// LS Electric XG5000 project: JG 비젼 프로그램
// PLC LSPLC
// module base 0 slot 0: 입출력 모듈:XBM-DN32H (DC 24V입력/TR 출력, 32점)

PROGRAM NewProgram (task: 스캔 프로그램)

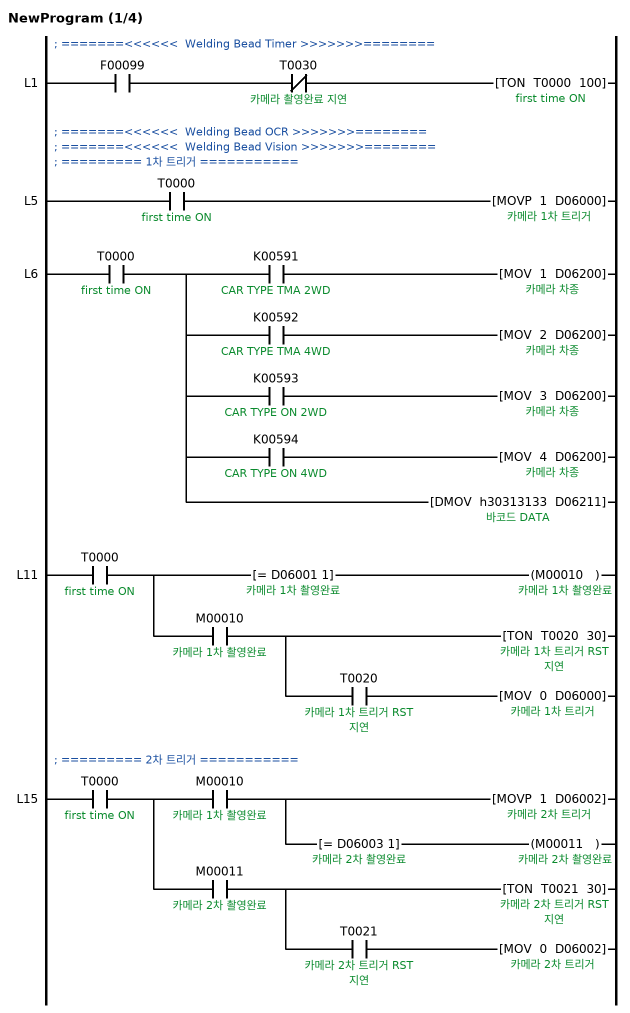
// =======<<<<<<  Welding Bead Timer >>>>>>>========
; L1
LOAD      F00099
AND NOT   T0030	// 카메라 촬영완료 지연
TON       T0000 100	// first time ON
// =======<<<<<<  Welding Bead OCR >>>>>>>========
// =======<<<<<<  Welding Bead Vision >>>>>>>========
// ========= 1차 트리거 ===========
; L5
LOAD      T0000	// first time ON
MOVP      1 D06000	// 카메라 1차 트리거
; L6
LOAD      T0000	// first time ON
MPUSH
AND       K00591	// CAR TYPE TMA 2WD
MOV       1 D06200	// 카메라 차종
MLOAD
AND       K00592	// CAR TYPE TMA 4WD
MOV       2 D06200	// 카메라 차종
MLOAD
AND       K00593	// CAR TYPE ON 2WD
MOV       3 D06200	// 카메라 차종
MLOAD
AND       K00594	// CAR TYPE ON 4WD
MOV       4 D06200	// 카메라 차종
MPOP
DMOV      h30313133 D06211	// 바코드 DATA
; L11
LOAD      T0000	// first time ON
MPUSH
AND=      D06001 1	// 카메라 1차 촬영완료
OUT       M00010	// 카메라 1차 촬영완료
MPOP
AND       M00010	// 카메라 1차 촬영완료
TON       T0020 30	// 카메라 1차 트리거 RST 지연
AND       T0020	// 카메라 1차 트리거 RST 지연
MOV       0 D06000	// 카메라 1차 트리거
// ========= 2차 트리거 ===========
; L15
LOAD      T0000	// first time ON
MPUSH
AND       M00010	// 카메라 1차 촬영완료
MOVP      1 D06002	// 카메라 2차 트리거
AND=      D06003 1	// 카메라 2차 촬영완료
OUT       M00011	// 카메라 2차 촬영완료
MPOP
AND       M00011	// 카메라 2차 촬영완료
TON       T0021 30	// 카메라 2차 트리거 RST 지연
AND       T0021	// 카메라 2차 트리거 RST 지연
MOV       0 D06002	// 카메라 2차 트리거

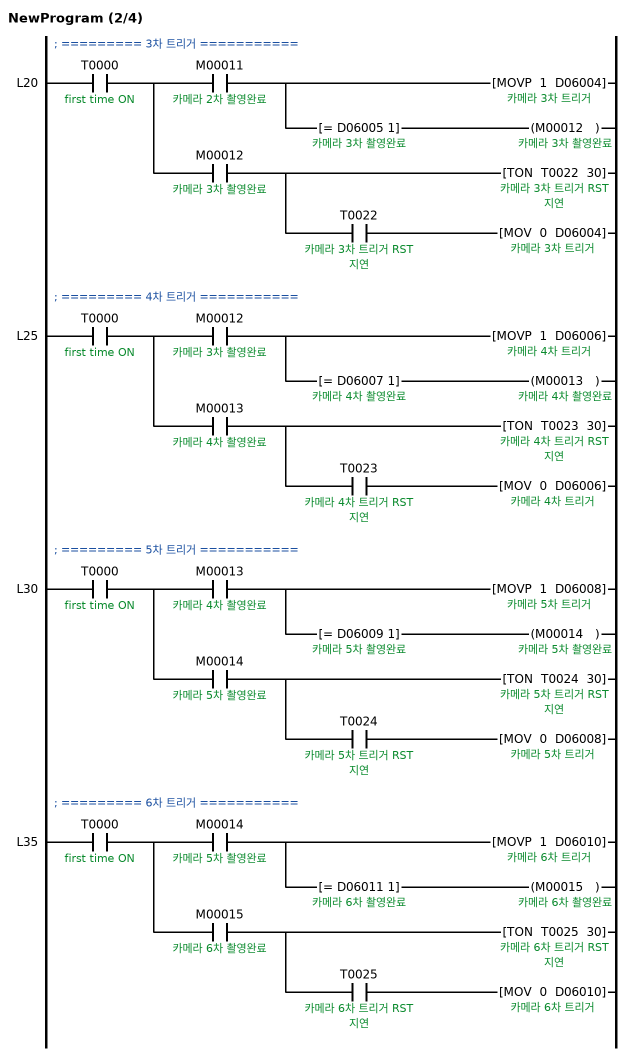
// ========= 3차 트리거 ===========
; L20
LOAD      T0000	// first time ON
MPUSH
AND       M00011	// 카메라 2차 촬영완료
MOVP      1 D06004	// 카메라 3차 트리거
AND=      D06005 1	// 카메라 3차 촬영완료
OUT       M00012	// 카메라 3차 촬영완료
MPOP
AND       M00012	// 카메라 3차 촬영완료
TON       T0022 30	// 카메라 3차 트리거 RST 지연
AND       T0022	// 카메라 3차 트리거 RST 지연
MOV       0 D06004	// 카메라 3차 트리거
// ========= 4차 트리거 ===========
; L25
LOAD      T0000	// first time ON
MPUSH
AND       M00012	// 카메라 3차 촬영완료
MOVP      1 D06006	// 카메라 4차 트리거
AND=      D06007 1	// 카메라 4차 촬영완료
OUT       M00013	// 카메라 4차 촬영완료
MPOP
AND       M00013	// 카메라 4차 촬영완료
TON       T0023 30	// 카메라 4차 트리거 RST 지연
AND       T0023	// 카메라 4차 트리거 RST 지연
MOV       0 D06006	// 카메라 4차 트리거
// ========= 5차 트리거 ===========
; L30
LOAD      T0000	// first time ON
MPUSH
AND       M00013	// 카메라 4차 촬영완료
MOVP      1 D06008	// 카메라 5차 트리거
AND=      D06009 1	// 카메라 5차 촬영완료
OUT       M00014	// 카메라 5차 촬영완료
MPOP
AND       M00014	// 카메라 5차 촬영완료
TON       T0024 30	// 카메라 5차 트리거 RST 지연
AND       T0024	// 카메라 5차 트리거 RST 지연
MOV       0 D06008	// 카메라 5차 트리거
// ========= 6차 트리거 ===========
; L35
LOAD      T0000	// first time ON
MPUSH
AND       M00014	// 카메라 5차 촬영완료
MOVP      1 D06010	// 카메라 6차 트리거
AND=      D06011 1	// 카메라 6차 촬영완료
OUT       M00015	// 카메라 6차 촬영완료
MPOP
AND       M00015	// 카메라 6차 촬영완료
TON       T0025 30	// 카메라 6차 트리거 RST 지연
AND       T0025	// 카메라 6차 트리거 RST 지연
MOV       0 D06010	// 카메라 6차 트리거

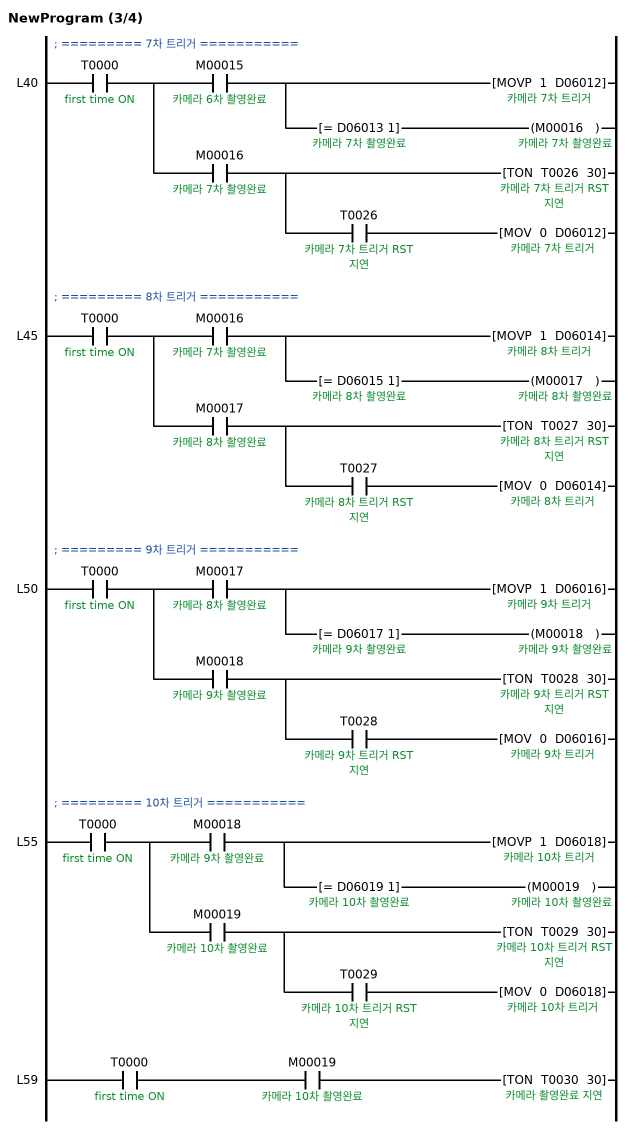
// ========= 7차 트리거 ===========
; L40
LOAD      T0000	// first time ON
MPUSH
AND       M00015	// 카메라 6차 촬영완료
MOVP      1 D06012	// 카메라 7차 트리거
AND=      D06013 1	// 카메라 7차 촬영완료
OUT       M00016	// 카메라 7차 촬영완료
MPOP
AND       M00016	// 카메라 7차 촬영완료
TON       T0026 30	// 카메라 7차 트리거 RST 지연
AND       T0026	// 카메라 7차 트리거 RST 지연
MOV       0 D06012	// 카메라 7차 트리거
// ========= 8차 트리거 ===========
; L45
LOAD      T0000	// first time ON
MPUSH
AND       M00016	// 카메라 7차 촬영완료
MOVP      1 D06014	// 카메라 8차 트리거
AND=      D06015 1	// 카메라 8차 촬영완료
OUT       M00017	// 카메라 8차 촬영완료
MPOP
AND       M00017	// 카메라 8차 촬영완료
TON       T0027 30	// 카메라 8차 트리거 RST 지연
AND       T0027	// 카메라 8차 트리거 RST 지연
MOV       0 D06014	// 카메라 8차 트리거
// ========= 9차 트리거 ===========
; L50
LOAD      T0000	// first time ON
MPUSH
AND       M00017	// 카메라 8차 촬영완료
MOVP      1 D06016	// 카메라 9차 트리거
AND=      D06017 1	// 카메라 9차 촬영완료
OUT       M00018	// 카메라 9차 촬영완료
MPOP
AND       M00018	// 카메라 9차 촬영완료
TON       T0028 30	// 카메라 9차 트리거 RST 지연
AND       T0028	// 카메라 9차 트리거 RST 지연
MOV       0 D06016	// 카메라 9차 트리거
// ========= 10차 트리거 ===========
; L55
LOAD      T0000	// first time ON
MPUSH
AND       M00018	// 카메라 9차 촬영완료
MOVP      1 D06018	// 카메라 10차 트리거
AND=      D06019 1	// 카메라 10차 촬영완료
OUT       M00019	// 카메라 10차 촬영완료
MPOP
AND       M00019	// 카메라 10차 촬영완료
TON       T0029 30	// 카메라 10차 트리거 RST 지연
AND       T0029	// 카메라 10차 트리거 RST 지연
MOV       0 D06018	// 카메라 10차 트리거
; L59
LOAD      T0000	// first time ON
AND       M00019	// 카메라 10차 촬영완료
TON       T0030 30	// 카메라 촬영완료 지연

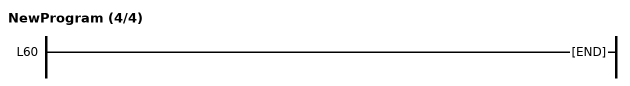
; L60
END

VARIABLES AND COMMENTS (devices not used above)
T0001	BIT/WORD	Welding Bead Trig ON
T0002	BIT/WORD	Trig OFF
P00020	BIT	OCR Trig
P00021	BIT	Visin Trig
T0010	BIT/WORD	OCR Trig time ready
M00020	BIT	OCR finish
T0005	BIT/WORD	Reset time